{attribute 'GeneratedUsingTerminal: EL3068-0000-0016'}
{attribute addProperty BoxType "EL3068-0000-0016"}
{attribute addProperty Id "EtcSlaveTerminalBaseAI_Standard_Channel_1AT %I*AI_Standard_Channel_EA9DF21E9AI_Standard_Channel_2AT %I*AI_Standard_Channel_EA9DF21E9AI_Standard_Channel_3AT %I*AI_Standard_Channel_EA9DF21E9AI_Standard_Channel_4AT %I*AI_Standard_Channel_EA9DF21E9AI_Standard_Channel_5AT %I*AI_Standard_Channel_EA9DF21E9AI_Standard_Channel_6AT %I*AI_Standard_Channel_EA9DF21E9AI_Standard_Channel_7AT %I*AI_Standard_Channel_EA9DF21E9AI_Standard_Channel_8AT %I*AI_Standard_Channel_EA9DF21E9WcStateAT %I*WcState_9091E0EB2InfoDataAT %I*InfoData_32EB74EA10"}
{attribute addProperty CRC "3665392119"}
{attribute addProperty Size "84"}
TYPE EL3068_DA7971F7 EXTENDS EtcSlaveTerminalBase :
STRUCT
	{attribute addProperty Name "AI_Standard_Channel_1"}
	AI_Standard_Channel_1 : AI_Standard_Channel_EA9DF21E;
	{attribute addProperty Name "AI_Standard_Channel_2"}
	AI_Standard_Channel_2 : AI_Standard_Channel_EA9DF21E;
	{attribute addProperty Name "AI_Standard_Channel_3"}
	AI_Standard_Channel_3 : AI_Standard_Channel_EA9DF21E;
	{attribute addProperty Name "AI_Standard_Channel_4"}
	AI_Standard_Channel_4 : AI_Standard_Channel_EA9DF21E;
	{attribute addProperty Name "AI_Standard_Channel_5"}
	AI_Standard_Channel_5 : AI_Standard_Channel_EA9DF21E;
	{attribute addProperty Name "AI_Standard_Channel_6"}
	AI_Standard_Channel_6 : AI_Standard_Channel_EA9DF21E;
	{attribute addProperty Name "AI_Standard_Channel_7"}
	AI_Standard_Channel_7 : AI_Standard_Channel_EA9DF21E;
	{attribute addProperty Name "AI_Standard_Channel_8"}
	AI_Standard_Channel_8 : AI_Standard_Channel_EA9DF21E;
	{attribute addProperty Name "WcState"}
	WcState : WcState_9091E0EB;
	{attribute addProperty Name "InfoData"}
	InfoData : InfoData_32EB74EA;
END_STRUCT
END_TYPE

(* stored: Version 1.2.0.0, ProductVersion 3.1.4024.9
   DUT EL3068_DA7971F7: Id {0f13f8a1-30dd-4d2c-82de-757f98ff2efc} *)
